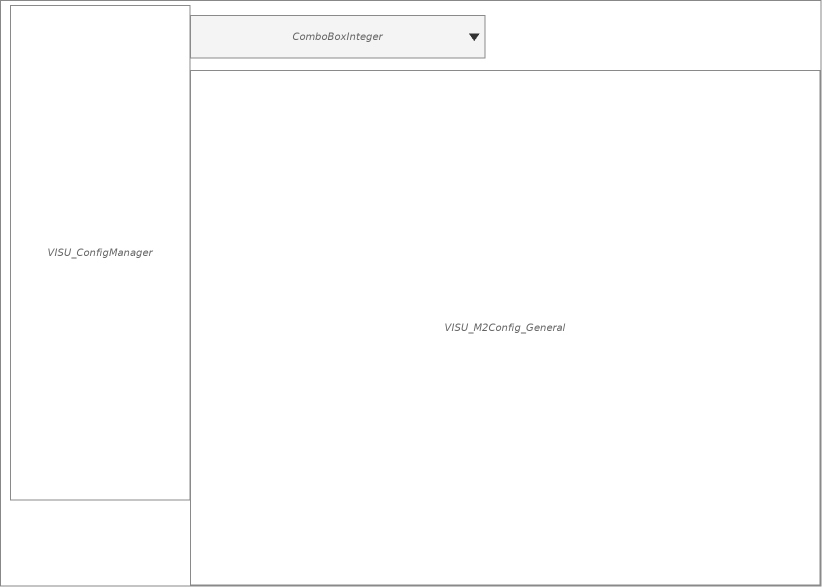
VISUALIZATION VISU_M2Config  // 822x587
VAR_IN_OUT
    editableConfig : M2Config;
	activeConfig : M2Config;
    mgr : ConfigManager;
    mgrWidget : ConfigManagerWidget;
    activeTab : INT;
	currentFocalStationPosition : INT;
END_VAR
    Frame (10,5 180x495)
        shows VISU_ConfigManager(mgr := mgr, widget := mgrWidget)
    ComboBoxInteger (190,15 295x43), variable: activeTab, text list: 'M2ConfigTabsTextList'
    Frame (190,70 630x515), frame switch variable: activeTab
        shows VISU_M2Config_General(editable := editableConfig, active := activeConfig)
        shows VISU_M2Config_PotentiometerAxis(editable := editableConfig.x, active := activeConfig.x)
        shows VISU_M2Config_PotentiometerAxis(editable := editableConfig.y, active := activeConfig.y)
        shows VISU_M2Config_ZAxis_General(editable := editableConfig.z, active := activeConfig.z)
        shows VISU_M2Config_ZAxis_Specific(editable := editableConfig.z, active := activeConfig.z)
        shows VISU_M2Config_PotentiometerAxis(editable := editableConfig.tiltX, active := activeConfig.tiltX)
        shows VISU_M2Config_PotentiometerAxis(editable := editableConfig.tiltY, active := activeConfig.tiltY)
        shows VISU_M2Config_ThermalFocus(currentPosition := currentFocalStationPosition, editable := editableConfig.thermalFocus, active := activeConfig.thermalFocus)
        shows VISU_M1Config_Axial_AverageForce(editable := editableConfig.axialSupport, active := activeConfig.axialSupport)
        shows VISU_MeasurementConfig(active := activeConfig.inclinometerVoltage, editable := editableConfig.inclinometerVoltage)
        p2735656198: currentFocalStationPosition
END_VISUALIZATION

(* stored: Version 1.1.0.1, ProductVersion 3.1.4019.2
   Visu VISU_M2Config: Id {4e289a0a-827c-4928-9eed-6e2009e2ad1a} *)
